ABB RAPID module: PointDesignationL.mod

MODULE PointDesignationL
     ! A point High enough so we prevent collision with right arm while counting the jars
    VAR robtarget HighPoint:=[[196.4363,403.2327,1110.746],[0.6038789,-0.03336211,0.3133152,0.7321549],[0,0,1,6],[-75.34075,9E+09,9E+09,9E+09,9E+09,9E+09]];

    ! Some points to move the jar from the corner of the orange station to it's place on the Black station
    CONST robtarget Mid_1:=[[554.8741,126.2235,262.6581],[0.1364978,0.4773159,0.8638731,-0.08521196],[0,0,1,4],[-114.2211,9E+09,9E+09,9E+09,9E+09,9E+09]];
    CONST robtarget Mid_2:=[[600.1525,126.022,252.2679],[0.2637084,-0.1631797,0.9305753,-0.194576],[0,-1,1,4],[-112.3011,9E+09,9E+09,9E+09,9E+09,9E+09]];
    CONST robtarget Mid_3:=[[477.903,13.94918,176.1371],[0.2316044,-0.2927044,0.7583622,-0.5343878],[0,-1,1,0],[-106.8015,9E+09,9E+09,9E+09,9E+09,9E+09]];
    CONST robtarget NearJar:=[[497.2253,-43.83931,99.90126],[0.3030509,-0.2875187,0.6406512,-0.6442509],[0,-1,1,0],[-97.47271,9E+09,9E+09,9E+09,9E+09,9E+09]];
    CONST robtarget AroundJar:=[[469.1461,57.8836,108.0806],[0.507771,-0.524942,0.4776943,-0.4882752],[0,2,1,0],[-104.2323,9E+09,9E+09,9E+09,9E+09,9E+09]];
    VAR   robtarget AroundJarTemp:=[[469.1461,57.8836,108.0806],[0.507771,-0.524942,0.4776943,-0.4882752],[0,2,1,0],[-104.2323,9E+09,9E+09,9E+09,9E+09,9E+09]];
    CONST robtarget AroundJar2:=[[542.9891,-82.73224,93.03219],[0.2985963,-0.3278764,0.6561838,-0.6105409],[0,-2,1,0],[-103.7693,9E+09,9E+09,9E+09,9E+09,9E+09]];
    CONST robtarget AroundJar2_whenreholdingB2ORNG:=[[469.1366,57.87084,77.23759],[0.507752,-0.5249463,0.4777046,-0.4882802],[0,2,1,0],[-108.5586,9E+09,9E+09,9E+09,9E+09,9E+09]];
    CONST robtarget AboveJar:=[[542.9725,-82.74228,181.6404],[0.2985748,-0.3278722,0.6561934,-0.6105433],[0,-2,1,0],[-103.7681,9E+09,9E+09,9E+09,9E+09,9E+09]];
    CONST robtarget AboveJarGripperClosed:=[[542.9536,-82.75277,130.0491],[0.2985461,-0.3278738,0.6561974,-0.6105522],[0,-2,1,0],[-103.7678,9E+09,9E+09,9E+09,9E+09,9E+09]];
    CONST robtarget AboveJarGripperClosedWithCover:=[[542.9536,-82.75277,133.5491],[0.2985461,-0.3278738,0.6561974,-0.6105522],[0,-2,1,0],[-103.7678,9E+09,9E+09,9E+09,9E+09,9E+09]];
    CONST robtarget Mid_4:=[[423.7296,10.00786,203.2406],[0.1999823,-0.2381262,0.7028769,-0.6397398],[0,-1,1,0],[-100.9323,9E+09,9E+09,9E+09,9E+09,9E+09]];
    CONST robtarget Mid_55:=[[399.0612,9.599308,227.3587],[0.09442355,0.1273759,0.7641647,-0.6252294],[0,-1,1,4],[-106.9641,9E+09,9E+09,9E+09,9E+09,9E+09]];
    CONST robtarget Mid_5:=[[294.4772,-31.24014,155.1631],[0.04340968,0.05411187,-0.7336182,0.6760117],[0,-1,1,0],[-88.41631,9E+09,9E+09,9E+09,9E+09,9E+09]];
    CONST robtarget Mid_6:=[[282.9144,9.219685,155.0747],[0.2976154,-0.2876453,-0.6585417,0.6284967],[0,0,1,0],[-89.4698,9E+09,9E+09,9E+09,9E+09,9E+09]];
    CONST robtarget AboveJarOnBlackStation:=[[300.4598,-108.7313,151.8091],[0.003938463,-0.003778499,-0.7494636,0.662023],[0,-1,1,0],[-106.3189,9E+09,9E+09,9E+09,9E+09,9E+09]];
    VAR  robtarget AboveJarOnBlackStationGripClosed:=[[297.6271,-108.8896,119.9425],[0.01007012,0.01952474,0.7378212,-0.6746386],[0,-1,1,0],[-86.27634,9E+09,9E+09,9E+09,9E+09,9E+09]];
    CONST robtarget AroundJarOnBlackStation:=[[300.4579,-108.7329,82.89008],[0.003940296,-0.003776616,-0.7494647,0.6620218],[0,-1,1,0],[-106.3195,9E+09,9E+09,9E+09,9E+09,9E+09]];
    VAR   robtarget AroundJarOnBlackStationTemp:=[[299.3644,-109.178,107.112],[0.02736216,0.0009125296,0.7063073,-0.7073758],[0,3,1,0],[-103.6667,9E+09,9E+09,9E+09,9E+09,9E+09]];
    CONST robtarget LiftComPos:=[[300.5263,-113.6614,67.16065],[0.002721211,-0.004066736,-0.7418641,0.6705323],[0,-1,1,0],[-105.7211,9E+09,9E+09,9E+09,9E+09,9E+09]];
    CONST robtarget JarLiftPositionSuc:=[[300.5102,-113.66146,171.1686],[0.0027393,-0.00406995,-0.7418638,0.6705326],[0,-1,1,0],[-105.7192,9E+09,9E+09,9E+09,9E+09,9E+09]];
    CONST robtarget JarLiftPositionFill:=[[300.4794,-113.6599,75.19614],[0.002774192,-0.004076869,-0.7418547,0.6705426],[0,-1,1,0],[-105.724,9E+09,9E+09,9E+09,9E+09,9E+09]];

    ! Points to take out nozzel if it get stucked (not emptied)
    CONST robtarget Mid_7:=[[370.2038,-32.87925,154.3524],[0.07468369,-0.01454502,-0.7141125,0.6958838],[0,-1,1,0],[-87.29718,9E+09,9E+09,9E+09,9E+09,9E+09]];
    CONST robtarget Mid_8:=[[298.1686,-36.30843,152.074],[0.4977928,-0.4529417,-0.5219991,0.5239877],[0,0,1,0],[-94.23718,9E+09,9E+09,9E+09,9E+09,9E+09]];
    CONST robtarget Mid_9:=[[186.6169,-50.05457,160.3339],[0.4734463,-0.4736413,-0.5224764,0.5277603],[0,0,1,0],[-91.6592,9E+09,9E+09,9E+09,9E+09,9E+09]];
    CONST robtarget Mid_10:=[[186.6181,-50.05502,140.333],[0.4734438,-0.4736429,-0.5224775,0.52776],[0,0,1,0],[-91.65925,9E+09,9E+09,9E+09,9E+09,9E+09]];
    CONST robtarget Mid_11:=[[186.5986,-50.04457,115.3932],[0.4734615,-0.4736465,-0.5224517,0.5277665],[0,0,1,0],[-102.8267,9E+09,9E+09,9E+09,9E+09,9E+09]];
    CONST robtarget Mid_12:=[[217.6369,12.78759,121.3941],[0.4734631,-0.4736456,-0.5224531,0.5277644],[0,0,1,0],[-102.8237,9E+09,9E+09,9E+09,9E+09,9E+09]];
    CONST robtarget Mid_13:=[[217.6287,67.39323,173.9318],[0.5328754,0.5396317,-0.4449165,-0.4763306],[0,0,-1,0],[-103.6128,9E+09,9E+09,9E+09,9E+09,9E+09]];
    CONST robtarget Mid_14:=[[74.23405,20.23655,236.8874],[0.5520811,0.5830978,-0.3836623,-0.4560775],[0,0,-1,0],[-103.5678,9E+09,9E+09,9E+09,9E+09,9E+09]];

    !points for opening jar lid by the right hand
    CONST robtarget OpenJarLidPoint:=[[438.2388,-72.98116,358.5548],[0.00297478,-0.001265666,0.7255163,-0.6881974],[1,3,1,4],[-105.4292,9E+09,9E+09,9E+09,9E+09,9E+09]];
    VAR   robtarget OpenJarLidPointTemp:=[[438.2388,-72.98116,358.5548],[0.00297478,-0.001265666,0.7255163,-0.6881974],[1,3,1,4],[-105.4292,9E+09,9E+09,9E+09,9E+09,9E+09]];
    VAR   robtarget Calibration_1:=[[299.3372,-109.1743,120.9315],[0.02733344,0.0009180704,0.7063079,-0.7073762],[0,3,1,0],[-103.664,9E+09,9E+09,9E+09,9E+09,9E+09]];

    !points For Held Jar in Hole Open And CLose
    CONST robtarget Held_AroundJarOnBlackStation:=[[299.3644,-109.178,82.112],[0.02736216,0.0009125296,0.7063073,-0.7073758],[0,3,1,0],[-103.6667,9E+09,9E+09,9E+09,9E+09,9E+09]];

    ! Point for the process: "PressToFill"
    VAR   robtarget PressToFill_1:=[[519.3063,24.34753,332.795],[0.02965483,-0.003819788,0.8239746,-0.5658373],[0,0,1,4],[-125.4765,9E+09,9E+09,9E+09,9E+09,9E+09]];
    VAR   robtarget PressToFill_2:=[[360.1791,-16.26686,468.5356],[0.02076531,0.07434192,-0.7122866,0.6976316],[0,1,-1,5],[-138.0943,9E+09,9E+09,9E+09,9E+09,9E+09]];
    VAR   robtarget PressToFill_3:=[[382.2147,-185.2293,384.7835],[0.04519064,0.01475611,-0.7181318,0.6942815],[0,1,-1,1],[-132.0769,9E+09,9E+09,9E+09,9E+09,9E+09]];
    VAR   robtarget PressToFill_4:=[[382.669,-190.6713,357.5512],[0.01741571,-0.005328834,-0.729151,0.6841105],[0,1,-1,1],[-128.3606,9E+09,9E+09,9E+09,9E+09,9E+09]];

!    VAR   robtarget PressToFill_33:=[[382.2147,-185.2293,384.7835],[0.04519064,0.01475611,-0.7181318,0.6942815],[0,1,-1,1],[-132.0769,9E+09,9E+09,9E+09,9E+09,9E+09]];
!    VAR   robtarget PressToFill_44:=[[382.2147,-185.2293,384.7835],[0.04519064,0.01475611,-0.7181318,0.6942815],[0,1,-1,1],[-132.0769,9E+09,9E+09,9E+09,9E+09,9E+09]];

    ! Point for the process: "PressToEmpty"
    VAR   robtarget PressToEmpty_1:=[[507.7589,-40.4017,439.5305],[0.05817171,-0.007579151,-0.7055872,0.7061907],[0,-1,1,4],[-114.2449,9E+09,9E+09,9E+09,9E+09,9E+09]];
    VAR   robtarget PressToEmpty_2:=[[409.6067,-92.53561,434.3977],[0.042205,0.04568755,-0.7053828,0.7060924],[0,-1,1,4],[-116.3767,9E+09,9E+09,9E+09,9E+09,9E+09]];
    VAR   robtarget PressToEmpty_3:=[[299.3842,-191.4462,440.1205],[0.05024188,-0.01052868,-0.7081174,0.7042263],[0,-1,1,4],[-127.8406,9E+09,9E+09,9E+09,9E+09,9E+09]];
    VAR   robtarget PressToEmpty_4:=[[293.096,-186.9429,416.2473],[0.07747618,-0.01482227,-0.7036266,0.706178],[0,-1,1,4],[-125.5751,9E+09,9E+09,9E+09,9E+09,9E+09]];

    ! Point for the process: "PressToDropNozzel"
    VAR   robtarget PressToDropNozzel_1:=[[461.1843,42.44297,476.7215],[0.06907275,-0.2256842,0.4523926,-0.8600212],[0,-1,1,4],[-111.1826,9E+09,9E+09,9E+09,9E+09,9E+09]];
    VAR   robtarget PressToDropNozzel_2:=[[372.7662,-47.38017,638.5932],[0.1921857,0.02402019,0.007670877,0.9810346],[0,-1,1,4],[-131.1653,9E+09,9E+09,9E+09,9E+09,9E+09]];
    VAR   robtarget PressToDropNozzel_3:=[[221.2352,-55.55732,540.6785],[0.4316385,-0.016244,0.01718291,0.9017367],[-2,-1,1,4],[-131.6921,9E+09,9E+09,9E+09,9E+09,9E+09]];
    VAR   robtarget PressToDropNozzel_4:=[[221.2341,-55.55516,525.4453],[0.4316393,-0.01624625,0.01718477,0.9017363],[-2,-1,1,4],[-131.6908,9E+09,9E+09,9E+09,9E+09,9E+09]];
! it was [233.9373,-54.62232,556.2691]

!    VAR   robtarget PressToDropNozzel_3:=[[256.4945,-57.30254,599.6307],[0.4860737,0.003330357,0.02276387,0.873615],[-1,-1,1,4],[-149.7138,9E+09,9E+09,9E+09,9E+09,9E+09]];
!    VAR   robtarget PressToDropNozzel_4:=[[233.9373,-54.62232,560.2691],[0.499564,-0.04660843,0.002983484,0.8650171],[-1,-1,1,4],[-152.252,9E+09,9E+09,9E+09,9E+09,9E+09]];

    VAR   robtarget TakeTheShit1:=[[634.1862,113.8697,192.1622],[0.3200693,-0.322839,0.6323941,-0.6272227],[-2,-1,1,4],[-99.01886,9E+09,9E+09,9E+09,9E+09,9E+09]];
    VAR   robtarget TakeTheShit2:=[[634.1827,-26.8355,192.1335],[0.3200635,-0.3228488,0.632426,-0.6271884],[-2,-2,1,4],[-104.1127,9E+09,9E+09,9E+09,9E+09,9E+09]];
    VAR   robtarget TakeTheShit3:=[[634.7637,-26.74809,100.5621],[0.3209175,-0.3231641,0.6328201,-0.6261914],[-2,-2,1,4],[-90.97301,9E+09,9E+09,9E+09,9E+09,9E+09]];
    VAR   robtarget TakeTheShit4:=[[233.9373,-54.62232,561.2691],[0.499564,-0.04660843,0.002983484,0.8650171],[-1,-1,1,4],[-152.252,9E+09,9E+09,9E+09,9E+09,9E+09]];
    VAR   robtarget TakeTheShit5:=[[233.9373,-54.62232,561.2691],[0.499564,-0.04660843,0.002983484,0.8650171],[-1,-1,1,4],[-152.252,9E+09,9E+09,9E+09,9E+09,9E+09]];
    VAR   robtarget TakeTheShit6:=[[233.9373,-54.62232,561.2691],[0.499564,-0.04660843,0.002983484,0.8650171],[-1,-1,1,4],[-152.252,9E+09,9E+09,9E+09,9E+09,9E+09]];
    VAR   robtarget TakeTheShit7:=[[233.9373,-54.62232,561.2691],[0.499564,-0.04660843,0.002983484,0.8650171],[-1,-1,1,4],[-152.252,9E+09,9E+09,9E+09,9E+09,9E+09]];
    VAR   robtarget TakeTheShit8:=[[233.9373,-54.62232,561.2691],[0.499564,-0.04660843,0.002983484,0.8650171],[-1,-1,1,4],[-152.252,9E+09,9E+09,9E+09,9E+09,9E+09]];

    !variables for pick_i_jar
    VAR robtarget temp11 := [[538.8864,-80.77894,221.9603],[0.006105556,-0.7083587,-0.7058232,-0.002063419],[0,1,0,0],[-143.5276,9E+09,9E+09,9E+09,9E+09,9E+09]];
    VAR robtarget temp22 := [[540.8173,-81.54366,142.0769],[0.01183519,-0.997568,-0.06846375,-0.005556368],[0,0,1,0],[-105.1789,9E+09,9E+09,9E+09,9E+09,9E+09]];
    VAR robtarget temp22_2 := [[538.8954,-80.79728,141.3239],[0.006108637,-0.708376,-0.7058056,-0.00213234],[0,1,0,0],[-143.5234,9E+09,9E+09,9E+09,9E+09,9E+09]];
    VAR robtarget temp33 := [[537.168,-23.01155,254.7484],[0.01269851,-0.9976652,-0.0668235,0.006131503],[0,1,1,0],[-137.7437,9E+09,9E+09,9E+09,9E+09,9E+09]];

    VAR robtarget temp111 := [[555.866,37.28145,260.7902],[0.003240219,0.515474,0.8375627,-0.1810106],[0,0,1,4],[-125.2034,9E+09,9E+09,9E+09,9E+09,9E+09]];

    ! points For EmptyJarInFunnel
    VAR robtarget EmptyJarInFunnel1 := [[542.9738,-82.7419,169.2278],[0.2985776,-0.3278701,0.6561945,-0.6105419],[0,-2,1,0],[-103.7685,9E+09,9E+09,9E+09,9E+09,9E+09]];
    VAR robtarget EmptyJarInFunnel2 := [[509.3815,-85.80142,333.4705],[0.2187517,-0.1670811,0.6963356,-0.6628335],[0,-1,1,4],[-120.4902,9E+09,9E+09,9E+09,9E+09,9E+09]];
    VAR robtarget EmptyJarInFunnel3 := [[522.1735,-69.93185,533.1119],[0.02160888,0.01557024,0.7216892,-0.6917046],[0,-1,0,4],[-131.8955,9E+09,9E+09,9E+09,9E+09,9E+09]];
    VAR robtarget EmptyJarInFunnel4 := [[579.168,-114.824,549.1523],[0.003460131,-0.01070567,0.7096465,-0.7044681],[0,-1,0,4],[-138.7548,9E+09,9E+09,9E+09,9E+09,9E+09]];
    VAR robtarget EmptyJarInFunnel5 := [[612.555,-124.0654,529.6832],[0.3797491,0.4447397,-0.5406042,0.604768],[0,-1,-1,4],[-138.8654,9E+09,9E+09,9E+09,9E+09,9E+09]];
    VAR jointtarget EmptyJarInFunnel6 := [[7.62782,-6.06867,-9.97302,-67.5133,48.472,-75.1432],[-11.3079,9E+09,9E+09,9E+09,9E+09,9E+09]];
    VAR robtarget EmptyJarInFunnel7 := [[639.8677,-123.5552,527.2377],[0.6505856,0.6549008,-0.1475849,0.3550521],[0,-1,-1,4],[-138.4516,9E+09,9E+09,9E+09,9E+09,9E+09]];
    VAR jointtarget EmptyJarInFunnel8 := [[7.62656,-4.88297,-12.1625,-71.4806,41.437,-137.477],[-12.4559,9E+09,9E+09,9E+09,9E+09,9E+09]];
!    VAR robtarget EmptyJarInFunnel1 := [[542.9738,-82.7419,169.2278],[0.2985776,-0.3278701,0.6561945,-0.6105419],[0,-2,1,0],[-103.7685,9E+09,9E+09,9E+09,9E+09,9E+09]];
!    VAR robtarget EmptyJarInFunnel2 := [[509.3815,-85.80142,333.4705],[0.2187517,-0.1670811,0.6963356,-0.6628335],[0,-1,1,4],[-120.4902,9E+09,9E+09,9E+09,9E+09,9E+09]];
!    VAR robtarget EmptyJarInFunnel3 := [[559.9003,-115.132,466.0972],[0.2435943,-0.18267,0.7031288,-0.6425756],[0,-1,1,4],[-135.0802,9E+09,9E+09,9E+09,9E+09,9E+09]];
!    VAR robtarget EmptyJarInFunnel4 := [[563.4829,-123.9325,453.4182],[0.1157927,-0.1737028,0.6953254,-0.6877077],[1,-1,1,4],[-101.6964,9E+09,9E+09,9E+09,9E+09,9E+09]];
!    VAR robtarget EmptyJarInFunnel5 := [[619.5551,-128.0116,495.3073],[0.09878946,0.2637755,-0.6589687,0.6974406],[1,-1,0,4],[-123.1754,9E+09,9E+09,9E+09,9E+09,9E+09]];
!    VAR jointtarget EmptyJarInFunnel6 := [[55.5188,-12.7313,-4.20476,-78.7748,51.5913,-66.4227],[-48.417,9E+09,9E+09,9E+09,9E+09,9E+09]];
!    VAR robtarget EmptyJarInFunnel7 := [[635.1245,-122.5695,495.139],[0.5098433,0.6154509,-0.3536144,0.4860419],[1,-1,-1,4],[-123.1736,9E+09,9E+09,9E+09,9E+09,9E+09]];
!    VAR jointtarget EmptyJarInFunnel8 := [[63.6341,-10.5993,-10.0918,-75.7709,53.0141,-103.894],[-55.7523,9E+09,9E+09,9E+09,9E+09,9E+09]];

    !points for TurnOnOffPump
    VAR robtarget TurnOnOffPump1 := [[526.153,38.09958,190.2548],[0.4197936,-0.5438984,0.5741237,-0.4453424],[0,-2,1,0],[-115.076,9E+09,9E+09,9E+09,9E+09,9E+09]];
    VAR robtarget TurnOnOffPump2 := [[606.993,68.08531,144.5578],[0.4903001,-0.5107632,0.4878295,-0.510636],[0,-2,1,0],[-115.457,9E+09,9E+09,9E+09,9E+09,9E+09]];
    VAR robtarget TurnOnOffPump3 := [[619.8333,69.28903,144.6728],[0.4774225,-0.5121061,0.5076672,-0.5020847],[0,-2,1,0],[-115.6113,9E+09,9E+09,9E+09,9E+09,9E+09]];
    VAR robtarget TurnOnOffPump4 := [[601.319,56.10294,144.9478],[0.4992474,-0.5128309,0.4744157,-0.5125294],[0,-2,1,0],[-117.0118,9E+09,9E+09,9E+09,9E+09,9E+09]];
    VAR robtarget TurnOnOffPump5 := [[620.4492,53.69436,144.059],[0.4864553,-0.5335312,0.4812441,-0.4971014],[0,-2,1,0],[-118.8294,9E+09,9E+09,9E+09,9E+09,9E+09]];

    !points to PutUsedFilterInPlate
    VAR robtarget PutUsedFilterInPlate1 := [[659.6804,294.5118,882.8145],[0.4583833,0.3134622,0.4479995,0.7006587],[1,1,1,4],[-84.16208,9E+09,9E+09,9E+09,9E+09,9E+09]];
    VAR robtarget PutUsedFilterInPlate2:= [[729.5361,316.8599,713.8459],[0.4743018,0.3458549,0.5544642,0.5899081],[-1,1,1,0],[-98.32429,9E+09,9E+09,9E+09,9E+09,9E+09]];
    VAR robtarget PutUsedFilterInPlate3 := [[627.6354,184.5434,403.376],[0.3160068,0.4302891,0.8267978,0.1771904],[-1,0,1,0],[-100.3993,9E+09,9E+09,9E+09,9E+09,9E+09]];
    VAR robtarget PutUsedFilterInPlate4 := [[693.8143,-76.36646,416.25],[0.4317127,0.4709601,0.739186,-0.2131308],[-1,0,1,4],[-144.9374,9E+09,9E+09,9E+09,9E+09,9E+09]];
    VAR robtarget PutUsedFilterInPlate5 := [[678.8909,-92.78428,400.3075],[0.4332832,0.4918353,0.7282541,-0.2000241],[-1,0,1,4],[-144.6771,9E+09,9E+09,9E+09,9E+09,9E+09]];
    VAR robtarget PutUsedFilterInPlate6 := [[675.0967,-96.8405,400.068],[0.4266095,0.459187,0.7422882,-0.2369805],[-1,0,1,4],[-144.0739,9E+09,9E+09,9E+09,9E+09,9E+09]];
    VAR robtarget PutUsedFilterInPlate7 := [[659.3943,-114.1817,416.0409],[0.433989,0.509519,0.6868571,-0.2833218],[-1,0,1,4],[-144.8195,9E+09,9E+09,9E+09,9E+09,9E+09]];
    VAR robtarget PutUsedFilterInPlate8 := [[660.7668,-108.0462,400.1559],[0.433766,0.5706262,0.6658683,-0.2070078],[-1,0,1,4],[-144.9431,9E+09,9E+09,9E+09,9E+09,9E+09]];
    VAR robtarget PutUsedFilterInPlate9_1 := [[653.9497,-117.6481,400.8684],[0.4377143,0.5433829,0.6762441,-0.2362946],[-1,0,1,4],[-144.7948,9E+09,9E+09,9E+09,9E+09,9E+09]];
    VAR robtarget PutUsedFilterInPlate9_2 := [[648.7224,-121.8801,400.2471],[0.4312582,0.5344699,0.6802632,-0.2561257],[-1,0,1,4],[-144.679,9E+09,9E+09,9E+09,9E+09,9E+09]];
    VAR robtarget PutUsedFilterInPlate9_3 := [[739.9978,-168.6412,416.739],[0.5754835,0.0372328,0.7205365,-0.3850449],[-2,0,1,5],[-176.9851,9E+09,9E+09,9E+09,9E+09,9E+09]];
    VAR robtarget PutUsedFilterInPlate9_4 := [[642.6837,-127.0515,399.5811],[0.4252243,0.525843,0.6833639,-0.2751133],[-1,0,1,4],[-144.6262,9E+09,9E+09,9E+09,9E+09,9E+09]];
    VAR robtarget PutUsedFilterInPlate10 := [[705.6974,15.20001,488.8885],[0.4072246,0.5465,0.6856457,-0.2557262],[-1,0,1,4],[-142.8558,9E+09,9E+09,9E+09,9E+09,9E+09]];
    VAR robtarget PutUsedFilterInPlate11 := [[540.3218,-77.23856,507.011],[0.6601061,0.1569522,0.7141562,-0.1720665],[-2,0,1,1],[-137.4751,9E+09,9E+09,9E+09,9E+09,9E+09]];
    VAR robtarget PutUsedFilterInPlate12 := [[520.2753,201.009,314.5901],[0.3981728,0.2501043,0.8246195,0.3144979],[-1,0,1,1],[-81.81605,9E+09,9E+09,9E+09,9E+09,9E+09]];
    VAR robtarget PutUsedFilterInPlate13 := [[685.7153,282.5469,791.6041],[0.3712364,0.4057675,0.3793415,0.7440674],[-1,0,1,1],[-85.34634,9E+09,9E+09,9E+09,9E+09,9E+09]];
    VAR robtarget PutUsedFilterInPlate14 := [[693.8467,-118.4703,438.5067],[0.5419858,0.1301268,0.7541113,-0.3473247],[-1,0,0,5],[-154.3998,9E+09,9E+09,9E+09,9E+09,9E+09]];

!    VAR robtarget PutUsedFilterInPlate1 := [[659.6804,294.5118,882.8145],[0.4583833,0.3134622,0.4479995,0.7006587],[1,1,1,4],[-84.16208,9E+09,9E+09,9E+09,9E+09,9E+09]];
!    VAR robtarget PutUsedFilterInPlate2:= [[729.5361,316.8599,713.8459],[0.4743018,0.3458549,0.5544642,0.5899081],[-1,1,1,0],[-98.32429,9E+09,9E+09,9E+09,9E+09,9E+09]];
!    VAR robtarget PutUsedFilterInPlate3 := [[627.6354,184.5434,403.376],[0.3160068,0.4302891,0.8267978,0.1771904],[-1,0,1,0],[-100.3993,9E+09,9E+09,9E+09,9E+09,9E+09]];
!    VAR robtarget PutUsedFilterInPlate4 := [[489.0176,30.28746,351.2016],[0.1877209,0.2861434,0.9252287,-0.1638134],[-1,0,1,0],[-103.505,9E+09,9E+09,9E+09,9E+09,9E+09]];
!    VAR robtarget PutUsedFilterInPlate5 := [[582.5636,-79.15766,464.9698],[0.4640646,0.1338722,0.8119465,-0.3278188],[-2,0,0,1],[-134.1977,9E+09,9E+09,9E+09,9E+09,9E+09]];
!    VAR robtarget PutUsedFilterInPlate6 := [[728.0447,-121.4309,437.2125],[0.5914922,0.08755949,0.7326388,-0.3251317],[-2,0,0,5],[-157.5888,9E+09,9E+09,9E+09,9E+09,9E+09]];
!    VAR robtarget PutUsedFilterInPlate7 := [[762.9458,-136.0914,431.3704],[0.5987817,0.06097189,0.7216019,-0.3421017],[-2,0,0,5],[-166.6636,9E+09,9E+09,9E+09,9E+09,9E+09]];
!    VAR robtarget PutUsedFilterInPlate8 := [[767.324,-138.3024,416.7769],[0.5755245,0.03726448,0.7204585,-0.3851265],[-2,1,0,5],[-176.9778,9E+09,9E+09,9E+09,9E+09,9E+09]];
!    VAR robtarget PutUsedFilterInPlate9_1 := [[753.6297,-152.0577,416.7436],[0.5754899,0.03723112,0.7205275,-0.3850524],[-2,0,0,5],[-176.9824,9E+09,9E+09,9E+09,9E+09,9E+09]];
!    VAR robtarget PutUsedFilterInPlate9_2 := [[749.1034,-159.2123,416.7399],[0.5754855,0.03723041,0.7205337,-0.3850474],[-2,0,0,5],[-176.9832,9E+09,9E+09,9E+09,9E+09,9E+09]];
!    VAR robtarget PutUsedFilterInPlate9_3 := [[739.9978,-168.6412,416.739],[0.5754835,0.0372328,0.7205365,-0.3850449],[-2,0,1,5],[-176.9851,9E+09,9E+09,9E+09,9E+09,9E+09]];
!    VAR robtarget PutUsedFilterInPlate9_4 := [[727.6697,-184.9677,416.7401],[0.575482,0.03723241,0.7205385,-0.3850435],[-2,0,1,5],[-176.9878,9E+09,9E+09,9E+09,9E+09,9E+09]];
!    VAR robtarget PutUsedFilterInPlate10 := [[716.1812,-180.2664,445.1152],[0.5987719,0.0609662,0.7216203,-0.3420811],[-2,0,1,5],[-166.6656,9E+09,9E+09,9E+09,9E+09,9E+09]];
!    VAR robtarget PutUsedFilterInPlate11 := [[540.3218,-77.23856,507.011],[0.6601061,0.1569522,0.7141562,-0.1720665],[-2,0,1,1],[-137.4751,9E+09,9E+09,9E+09,9E+09,9E+09]];
!    VAR robtarget PutUsedFilterInPlate12 := [[520.2753,201.009,314.5901],[0.3981728,0.2501043,0.8246195,0.3144979],[-1,0,1,1],[-81.81605,9E+09,9E+09,9E+09,9E+09,9E+09]];
!    VAR robtarget PutUsedFilterInPlate13 := [[685.7153,282.5469,791.6041],[0.3712364,0.4057675,0.3793415,0.7440674],[-1,0,1,1],[-85.34634,9E+09,9E+09,9E+09,9E+09,9E+09]];
!    VAR robtarget PutUsedFilterInPlate14 := [[693.8467,-118.4703,438.5067],[0.5419858,0.1301268,0.7541113,-0.3473247],[-1,0,0,5],[-154.3998,9E+09,9E+09,9E+09,9E+09,9E+09]];

    !Points for TwoPartsRemovingFilter
    VAR robtarget TwoPartsRemovingFilter1 := [[693.8467,-118.4703,438.5067],[0.5419858,0.1301268,0.7541113,-0.3473247],[-1,0,0,5],[-154.3998,9E+09,9E+09,9E+09,9E+09,9E+09]];
    VAR robtarget TwoPartsRemovingFilter2 := [[693.8467,-118.4703,438.5067],[0.5419858,0.1301268,0.7541113,-0.3473247],[-1,0,0,5],[-154.3998,9E+09,9E+09,9E+09,9E+09,9E+09]];
    VAR robtarget TwoPartsRemovingFilter3 := [[693.8467,-118.4703,438.5067],[0.5419858,0.1301268,0.7541113,-0.3473247],[-1,0,0,5],[-154.3998,9E+09,9E+09,9E+09,9E+09,9E+09]];
    VAR robtarget TwoPartsRemovingFilter4 := [[693.8467,-118.4703,438.5067],[0.5419858,0.1301268,0.7541113,-0.3473247],[-1,0,0,5],[-154.3998,9E+09,9E+09,9E+09,9E+09,9E+09]];
    VAR robtarget TwoPartsRemovingFilter5 := [[693.8467,-118.4703,438.5067],[0.5419858,0.1301268,0.7541113,-0.3473247],[-1,0,0,5],[-154.3998,9E+09,9E+09,9E+09,9E+09,9E+09]];
    VAR robtarget TwoPartsRemovingFilter6 := [[693.8467,-118.4703,438.5067],[0.5419858,0.1301268,0.7541113,-0.3473247],[-1,0,0,5],[-154.3998,9E+09,9E+09,9E+09,9E+09,9E+09]];
    VAR robtarget TwoPartsRemovingFilter7 := [[693.8467,-118.4703,438.5067],[0.5419858,0.1301268,0.7541113,-0.3473247],[-1,0,0,5],[-154.3998,9E+09,9E+09,9E+09,9E+09,9E+09]];
    VAR robtarget TwoPartsRemovingFilter8 := [[693.8467,-118.4703,438.5067],[0.5419858,0.1301268,0.7541113,-0.3473247],[-1,0,0,5],[-154.3998,9E+09,9E+09,9E+09,9E+09,9E+09]];

    ! Points for OpenLock
    VAR robtarget OpenLock1 := [[444.457,57.70416,428.058],[0.03391873,-0.7404301,-0.6687696,0.05796584],[0,0,1,4],[-130.1532,9E+09,9E+09,9E+09,9E+09,9E+09]];
    VAR robtarget OpenLock2 := [[395.5481,-18.01055,662.0746],[0.2859399,0.623473,0.6130692,-0.3920025],[0,0,0,4],[-175.4325,9E+09,9E+09,9E+09,9E+09,9E+09]];
    VAR robtarget OpenLock3 := [[140.0657,208.4361,815.2481],[0.7192939,0.5369508,0.3359022,-0.2854294],[-1,0,0,4],[-173.6447,9E+09,9E+09,9E+09,9E+09,9E+09]];
    VAR robtarget OpenLock4 := [[5.191932,227.3297,792.3666],[0.7067034,0.6950218,-0.1054061,-0.08002785],[-1,0,1,4],[-177.0995,9E+09,9E+09,9E+09,9E+09,9E+09]];
    VAR robtarget OpenLock5 := [[-0.2072967,211.4303,796.5233],[0.6647114,0.7327977,-0.1080445,-0.0974303],[0,0,1,4],[-174.9861,9E+09,9E+09,9E+09,9E+09,9E+09]];
    VAR robtarget OpenLock6 := [[18.56533,206.4703,803.4706],[0.5342917,0.7544999,-0.1925943,-0.3288917],[0,0,1,4],[174.4749,9E+09,9E+09,9E+09,9E+09,9E+09]];
    VAR robtarget OpenLock7 := [[26.01069,197.7451,805.874],[0.5572425,0.7538844,-0.1712465,-0.3030078],[0,0,1,4],[174.3886,9E+09,9E+09,9E+09,9E+09,9E+09]];
    VAR robtarget OpenLock8 := [[64.29567,196.4137,796.8171],[0.593984,0.7749357,-0.1077863,-0.1871893],[0,0,1,4],[174.6816,9E+09,9E+09,9E+09,9E+09,9E+09]];
    VAR robtarget OpenLock9 := [[141.9606,292.9066,771.1875],[0.6093736,0.7831045,0.0007116533,-0.1241395],[-1,0,1,4],[168.4337,9E+09,9E+09,9E+09,9E+09,9E+09]];
    VAR robtarget OpenDoor1 := [[9.252483,190.8387,946.1296],[0.5472443,0.4799712,-0.5484715,0.4114976],[0,0,2,4],[-170.3192,9E+09,9E+09,9E+09,9E+09,9E+09]];
    VAR robtarget OpenDoor2 := [[74.19608,109.5013,916.4993],[0.4329654,0.6321019,-0.5041171,0.398565],[0,0,2,4],[-170.9254,9E+09,9E+09,9E+09,9E+09,9E+09]];
    VAR robtarget OpenDoor3 := [[89.49784,107.546,916.007],[0.5552816,0.796127,-0.1462974,0.1908958],[0,0,1,4],[-171.0104,9E+09,9E+09,9E+09,9E+09,9E+09]];
    VAR robtarget OpenDoor4 := [[151.8988,-17.92328,903.7396],[0.6081921,0.7752277,-0.08229822,0.1495035],[0,0,1,4],[-165.7217,9E+09,9E+09,9E+09,9E+09,9E+09]];
    VAR robtarget OpenDoor5 := [[128.8867,-153.3557,902.482],[0.6733187,0.7204248,-0.1633569,0.03073454],[0,0,1,4],[172.9512,9E+09,9E+09,9E+09,9E+09,9E+09]];
    VAR robtarget OpenDoor6 := [[89.68587,-220.5704,903.4578],[0.6246813,0.7343436,0.08674885,-0.250973],[0,0,1,4],[-177.4566,9E+09,9E+09,9E+09,9E+09,9E+09]];
    VAR robtarget OpenDoor7 := [[75.34122,-242.0442,913.9324],[0.6577976,0.7158023,-0.01540221,-0.2338637],[0,0,1,4],[-178.3179,9E+09,9E+09,9E+09,9E+09,9E+09]];
    VAR robtarget OpenDoor8 := [[31.01233,-264.0635,919.3221],[0.6670828,0.6893996,-0.1408893,-0.2447015],[0,-1,1,4],[-174.4533,9E+09,9E+09,9E+09,9E+09,9E+09]];
    VAR robtarget OpenDoor9 := [[-22.00384,-264.0953,915.5707],[0.6219023,0.6198655,-0.2969985,-0.375228],[1,-1,2,4],[-179.6873,9E+09,9E+09,9E+09,9E+09,9E+09]];

    VAR num botNumber;

    VAR robtarget Error_TurnCtfg1 := [[170.2733,577.2457,243.9488],[0.00239963,0.3935039,-0.9193189,0.001257257],[1,-1,1,0],[-71.50956,9E+09,9E+09,9E+09,9E+09,9E+09]];
    VAR robtarget Error_TurnCtfg2 := [[-22.00384,-264.0953,915.5707],[0.6219023,0.6198655,-0.2969985,-0.375228],[1,-1,2,4],[-179.6873,9E+09,9E+09,9E+09,9E+09,9E+09]];
    VAR robtarget Error_TurnCtfg3 := [[-22.00384,-264.0953,915.5707],[0.6219023,0.6198655,-0.2969985,-0.375228],[1,-1,2,4],[-179.6873,9E+09,9E+09,9E+09,9E+09,9E+09]];

    VAR jointtarget shakeTubeClosed2 := [[3.84446,22.2276,18.0538,-143.954,79.6974,107.872],[24.8287,9E+09,9E+09,9E+09,9E+09,9E+09]];
    VAR jointtarget shakeTubeClosed3 := [[3.84446,22.2276,18.0538,-143.954,79.6974,107.872],[24.8287,9E+09,9E+09,9E+09,9E+09,9E+09]];

    VAR robtarget TightEquipping_1 := [[534.7612,-66.24588,448.1762],[0.0492238,0.994812,-0.08824188,0.01181438],[0,1,2,4],[-162.2959,9E+09,9E+09,9E+09,9E+09,9E+09]];
    VAR robtarget TightEquipping_2 := [[542.2573,-87.87419,378.4257],[0.01285309,-0.9964926,0.08052952,0.01876991],[0,1,1,0],[-166.3403,9E+09,9E+09,9E+09,9E+09,9E+09]];
    VAR robtarget TightEquipping_2_2 := [[541.673,-87.16678,340.6087],[0.004533053,0.9957977,-0.09128092,0.005848722],[0,1,1,0],[-156.5342,9E+09,9E+09,9E+09,9E+09,9E+09]];
    VAR robtarget TightEquipping_3 := [[541.676,-87.17374,325.7926],[0.004511012,0.9957966,-0.09129214,0.005883972],[0,1,1,0],[-156.5287,9E+09,9E+09,9E+09,9E+09,9E+09]];

    VAR robtarget PlaceFilterT1 := [[611.5538,188.9556,446.433],[0.4805578,-0.4926687,0.4904753,-0.53458],[0,-2,1,4],[-126.2647,9E+09,9E+09,9E+09,9E+09,9E+09]];
    VAR robtarget PlaceFilterT2 := [[630.3646,-3.842554,422.7774],[0.4727144,0.4460948,0.6930832,-0.3117309],[0,-1,1,4],[-127.4054,9E+09,9E+09,9E+09,9E+09,9E+09]];
    VAR robtarget PlaceFilterT3 := [[-53.30389,101.794,388.8003],[0.4561347,0.4681619,0.7094583,-0.2635043],[0,-1,1,4],[-128.3209,9E+09,9E+09,9E+09,9E+09,9E+09]];
    VAR robtarget PlaceFilterT4 := [[-47.41281,92.84719,385.8619],[0.4570908,0.4124958,0.7358824,-0.2817665],[0,-1,1,4],[-128.1705,9E+09,9E+09,9E+09,9E+09,9E+09]];
    VAR robtarget PlaceFilterT5 := [[-34.62054,96.09262,371.6744],[0.5329425,0.4002055,0.6885161,-0.2859257],[0,-1,2,4],[-123.7589,9E+09,9E+09,9E+09,9E+09,9E+09]];
    VAR robtarget PlaceFilterT6 := [[-51.12422,93.0301,363.8972],[0.5497394,0.4443694,0.6214367,-0.3378446],[0,-1,2,4],[-120.1642,9E+09,9E+09,9E+09,9E+09,9E+09]];
    VAR robtarget PlaceFilterT7 := [[-50.19769,79.45396,361.1102],[0.5492472,0.4124961,0.6310747,-0.3604431],[0,-1,2,4],[-120.3211,9E+09,9E+09,9E+09,9E+09,9E+09]];
    VAR robtarget PlaceFilterAbovePlate := [[-62.8074,56.11432,382.8491],[0.5123566,0.4925491,0.6392291,-0.2937214],[0,-1,2,4],[-127.7035,9E+09,9E+09,9E+09,9E+09,9E+09]];
    VAR robtarget PlaceFilterNearPlate := [[-45.5563,88.54259,396.3635],[0.5607795,0.3929399,0.6269881,-0.3714975],[0,-1,2,4],[-122.5446,9E+09,9E+09,9E+09,9E+09,9E+09]];
    VAR robtarget AwayFromPlate := [[-75.52215,109.7407,413.4696],[0.4992928,0.4945384,0.641796,-0.3069795],[0,-1,1,4],[-126.8027,9E+09,9E+09,9E+09,9E+09,9E+09]];
    VAR robtarget AboveTweezers := [[554.6125,187.2478,347.3214],[0.009141128,0.004833775,0.9999462,-0.0008103135],[1,0,0,4],[-91.82567,9E+09,9E+09,9E+09,9E+09,9E+09]];

    VAR robtarget TweezHelp1 := [[511.9012,185.3691,245.455],[0.2224359,-0.002102946,0.9749377,0.003773012],[2,-1,1,1],[-132.7921,9E+09,9E+09,9E+09,9E+09,9E+09]];

    VAR robtarget AboveTweezersReorient := [[558.8926,186.2785,147.8935],[0.221747,-0.007361691,0.975073,0.002584573],[1,0,1,1],[-112.0385,9E+09,9E+09,9E+09,9E+09,9E+09]];

    VAR robtarget AroundTweezersClose := [[567.4321,186.5397,219.4024],[0.4232465,0.006302222,0.9059864,0.003347539],[1,0,0,5],[-103.7297,9E+09,9E+09,9E+09,9E+09,9E+09]];
    VAR robtarget AroundTweezers := [[558.8488,186.2694,147.8692],[0.4070934,-0.004760375,0.9133582,0.005390874],[1,0,0,1],[-110.2104,9E+09,9E+09,9E+09,9E+09,9E+09]];
    VAR robtarget AroundTweezersGrip := [[558.4938,186.8937,134.9628],[0.009139122,0.00481677,0.9999463,-0.0008170585],[2,0,0,4],[-91.89567,9E+09,9E+09,9E+09,9E+09,9E+09]];


    VAR robtarget demonL1 := [[522.76,101.508,370.2567],[0.6395594,0.6600569,0.2778583,0.279434],[0,1,1,5],[-103.3218,9E+09,9E+09,9E+09,9E+09,9E+09]];
    VAR robtarget demonL2 := [[751.3519,323.1772,506.6777],[0.4281275,-0.6848934,0.4830146,-0.3381196],[0,0,-1,4],[-95.64716,9E+09,9E+09,9E+09,9E+09,9E+09]];


    VAR robtarget PickAndPlaceDoneAnalysisJars1 := [[537.182,-23.00752,254.7764],[0.01267209,-0.9976645,-0.06683949,0.006113062],[0,1,1,0],[-137.745,9E+09,9E+09,9E+09,9E+09,9E+09]];
    VAR robtarget PickAndPlaceDoneAnalysisJars2 := [[570.4759,125.5156,319.4925],[0.02538738,-0.9760913,-0.2154495,-0.0135202],[0,1,1,4],[-128.7419,9E+09,9E+09,9E+09,9E+09,9E+09]];
    VAR robtarget PickAndPlaceDoneAnalysisJars3 := [[540.7717,196.3669,306.0183],[0.2542661,-0.8990465,-0.2785631,-0.2224113],[0,1,1,4],[-127.332,9E+09,9E+09,9E+09,9E+09,9E+09]];
    VAR robtarget PickAndPlaceDoneAnalysisJars4 := [[525.423,188.4654,277.9547],[0.3815894,-0.5806725,0.5867504,-0.415852],[1,2,1,4],[-98.31242,9E+09,9E+09,9E+09,9E+09,9E+09]];
    VAR robtarget PickAndPlaceDoneAnalysisJars5 := [[561.7964,206.3241,252.4906],[0.3828885,-0.6013064,0.5689505,-0.4100272],[1,2,1,4],[-99.68642,9E+09,9E+09,9E+09,9E+09,9E+09]];
    VAR robtarget PickAndPlaceDoneAnalysisJars6 := [[655.5176,208.3491,209.3318],[0.3739311,-0.6130069,0.5491101,-0.4276402],[1,2,1,0],[-105.7962,9E+09,9E+09,9E+09,9E+09,9E+09]];
    VAR robtarget PickAndPlaceDoneAnalysisJars7 := [[525.423,188.4654,277.9547],[0.3815894,-0.5806725,0.5867504,-0.415852],[1,2,1,4],[-98.31242,9E+09,9E+09,9E+09,9E+09,9E+09]];
    VAR robtarget PickAndPlaceDoneAnalysisJars8 := [[587.5679,152.8891,234.2181],[0.4177889,-0.5915911,0.5426972,-0.4253847],[1,2,1,4],[-107.021,9E+09,9E+09,9E+09,9E+09,9E+09]];
    VAR robtarget PickAndPlaceDoneAnalysisJars9 := [[656.011,157.5958,208.3058],[0.4112938,-0.5956156,0.5396773,-0.4299162],[1,2,1,0],[-112.4389,9E+09,9E+09,9E+09,9E+09,9E+09]];
    VAR robtarget PickAndPlaceDoneAnalysisJars10 := [[525.423,188.4654,277.9547],[0.3815894,-0.5806725,0.5867504,-0.415852],[1,2,1,4],[-98.31242,9E+09,9E+09,9E+09,9E+09,9E+09]];

    !Points To Pick Jars From Their Station
    CONST robtarget Jar_i:=[[578.174,59.39053,136.758],[0.004271943,-0.9989691,-0.04503585,0.003779688],[-1,1,1,4],[-140.1295,9E+09,9E+09,9E+09,9E+09,9E+09]];
    VAR robtarget Jar_i_changing:=[[576.117,59.88061,138.5151],[0.001168195,-0.4148987,-0.9098623,0.002880127],[0,1,0,0],[-123.9672,9E+09,9E+09,9E+09,9E+09,9E+09]];
    CONST robtarget point_i:=[[576.1957,57.64332,274.0359],[0.0009735118,0.9987404,0.04927012,-0.009441065],[-1,1,1,4],[-140.0888,9E+09,9E+09,9E+09,9E+09,9E+09]];
    VAR robtarget point_i_changing:=[[575.8237,59.84186,160.0466],[0.001460813,-0.4148932,-0.9098634,0.003189074],[0,1,0,0],[-123.9444,9E+09,9E+09,9E+09,9E+09,9E+09]];
    ! Main MidPoint Of The System, abbreviated as "MMP"
    CONST robtarget MainMidPoint:=[[391.3701,138.0784,287.818],[0.01673144,-0.6788682,-0.7340627,-0.003146656],[0,0,1,4],[-105.6234,9E+09,9E+09,9E+09,9E+09,9E+09]];

    ! Centrifuge Center
    CONST robtarget CentrifugeCenter:=[[170.9407,572.1271,375.2909],[0.002034158,0.3950241,-0.9186674,0.001424496],[1,-1,1,0],[53.36959,9E+09,9E+09,9E+09,9E+09,9E+09]];

    ! Home of Left Arm
    CONST robtarget LeftArmHome:=[[-25.10183,35.87066,242.0362],[0.5241755,-0.456079,-0.4959679,0.5208146],[0,0,1,0],[-100.0034,9E+09,9E+09,9E+09,9E+09,9E+09]];
    CONST robtarget LeftArmHome2:=[[91.8348,42.58352,228.3557],[0.5194696,-0.447556,-0.5231068,0.5061662],[0,0,1,0],[-108.0553,9E+09,9E+09,9E+09,9E+09,9E+09]];

    ! Two points to rotate the Centrifuge rotor (axis)
    VAR jointtarget JointValuesAtRotationPoint := [[122.239,29.7559,-19.7606,-66.2785,71.2014,156.395],[3.56826,9E+09,9E+09,9E+09,9E+09,9E+09]];
    VAR jointtarget JointValuesAboveRotationPoint := [[119.561,28.2938,-22.0489,-67.2533,80.1595,74.3327],[13.3094,9E+09,9E+09,9E+09,9E+09,9E+09]];
    VAR jointtarget ApproachingPointAboveBlackSpot := [[106.568,30.0729,-17.8489,-77.2586,78.6877,35.8075],[28.6868,9E+09,9E+09,9E+09,9E+09,9E+09]];
    VAR jointtarget ApproachingPointAboveBlackSpot_2 := [[108.064,28.8972,-18.132,-76.5745,81.6513,35.4804],[29.6382,9E+09,9E+09,9E+09,9E+09,9E+09]];

    ! Points On The Path From MainMidPoint To Open Lid
    CONST robtarget FromMainMidPointToOpenLid1:=[[555.6271,255.7578,292.2513],[0.05483364,-0.590986,-0.8012478,-0.07570177],[0,0,1,4],[-108.0667,9E+09,9E+09,9E+09,9E+09,9E+09]];
    CONST robtarget FromMainMidPointToOpenLid2:=[[530.2897,361.5968,268.8058],[0.1494315,-0.5993652,-0.7668331,-0.174352],[0,1,1,4],[-100.0325,9E+09,9E+09,9E+09,9E+09,9E+09]];
    CONST robtarget FromMainMidPointToOpenLid3:=[[515.9312,467.775,263.5276],[0.03093584,0.1698122,0.935509,0.3082689],[0,0,0,4],[-80.93092,9E+09,9E+09,9E+09,9E+09,9E+09]];
    CONST robtarget FromMainMidPointToOpenLid4:=[[505.7648,470.2841,261.1846],[0.002194192,0.1675383,0.9377017,0.3043708],[0,0,0,4],[-81.04429,9E+09,9E+09,9E+09,9E+09,9E+09]];
    CONST robtarget StuckLidOpen1:=[[511.3714,387.8458,287.1512],[0.02826629,0.1820043,-0.9136657,-0.3623403],[1,0,0,4],[-71.72851,9E+09,9E+09,9E+09,9E+09,9E+09]];
    CONST robtarget StuckLidOpen2:=[[434.6936,360.7884,304.8413],[0.2318009,0.3091172,-0.7584912,-0.5247914],[2,0,0,4],[-53.44424,9E+09,9E+09,9E+09,9E+09,9E+09]];
    CONST robtarget StuckLidOpen3:=[[357.247,420.9841,302.484],[0.1812195,0.3416057,-0.7585484,-0.5244706],[2,0,0,4],[-46.24845,9E+09,9E+09,9E+09,9E+09,9E+09]];
    CONST robtarget StuckLidOpen4:=[[358.1856,425.442,389.0001],[0.04476143,0.5862212,-0.7014162,-0.4029348],[1,0,0,4],[-38.2786,9E+09,9E+09,9E+09,9E+09,9E+09]];
    CONST robtarget StuckLidOpen5:=[[332.1754,461.2852,492.5867],[0.08736742,-0.7816244,0.5270592,0.3219299],[1,0,0,4],[-8.962341,9E+09,9E+09,9E+09,9E+09,9E+09]];
    CONST robtarget StuckLidOpen6:=[[293.2359,466.8463,540.8222],[0.1258348,-0.8279678,0.4477544,0.3132907],[1,0,0,4],[5.271636,9E+09,9E+09,9E+09,9E+09,9E+09]];
    CONST robtarget StuckLidOpen7:=[[261.7409,484.2215,580.4375],[0.1996818,-0.8599576,0.3676526,0.2922871],[1,0,0,4],[19.18535,9E+09,9E+09,9E+09,9E+09,9E+09]];
    CONST robtarget StuckLidOpen8:=[[483.4654,510.2447,469.6231],[0.7102606,-0.5688905,0.09371739,-0.4038694],[0,2,1,4],[-106.5761,9E+09,9E+09,9E+09,9E+09,9E+09]];

    ! Points On The Path From MainMidPoint To the center of Centrifuge
    CONST robtarget FromMainMidPointToMidCtfg3:=[[450.2527,158.2175,451.6961],[0.01001458,0.6602603,0.7509692,-0.001124735],[1,0,1,4],[-82.61719,9E+09,9E+09,9E+09,9E+09,9E+09]];
    CONST robtarget FromMainMidPointToMidCtfg4:=[[323.9157,496.4598,484.945],[0.01640962,-0.2539656,0.9670679,-0.003446209],[1,-1,1,4],[20.83673,9E+09,9E+09,9E+09,9E+09,9E+09]];
    CONST robtarget FromMainMidPointToMidCtfg5:=[[210.4415,548.9407,460.6745],[0.001568333,0.3650672,-0.9308972,-0.01240387],[1,-1,1,0],[56.035,9E+09,9E+09,9E+09,9E+09,9E+09]];

    ! Points On The Path From MidCtfg To 0_angleHole
    CONST robtarget FromMidCtfg1To_0_angleHole1:=[[135.2472,548.4155,379.5739],[0.1102394,0.4009789,-0.9091622,0.02207327],[1,-1,1,0],[56.79922,9E+09,9E+09,9E+09,9E+09,9E+09]];
    CONST robtarget FromMidCtfg1To_0_angleHole2:=[[137.767,549.8556,345.9562],[0.1433132,0.3114628,-0.9385209,0.04038253],[1,-1,1,0],[30.70798,9E+09,9E+09,9E+09,9E+09,9E+09]];
    VAR   robtarget FromMidCtfg1To_0_angleHole3:=[[110.7217,535.2574,266.8914],[0.1269187,0.3825924,-0.9146844,0.02944688],[1,-1,1,0],[-98.19913,9E+09,9E+09,9E+09,9E+09,9E+09]];
    VAR   robtarget FromMidCtfg1To_0_angleHole3_New:=[[111.789,535.7997,267.7856],[0.1274696,0.3878011,-0.9109861,0.05887322],[1,-1,1,0],[-105.3579,9E+09,9E+09,9E+09,9E+09,9E+09]];

    ! Points On The Path From MidCtfg To 180_angleHole
    CONST robtarget FromMidCtfg1To_180_angleHole1:=[[204.7944,601.0034,381.2636],[0.1095933,-0.3805622,0.917484,0.03721399],[1,-1,1,0],[51.17107,9E+09,9E+09,9E+09,9E+09,9E+09]];
    CONST robtarget FromMidCtfg1To_180_angleHole2:=[[209.0023,611.7137,346.9704],[0.1469437,-0.2921586,0.9440864,0.04185314],[1,-1,1,0],[29.28295,9E+09,9E+09,9E+09,9E+09,9E+09]];
    VAR   robtarget FromMidCtfg1To_180_angleHole3:=[[223.1574,615.9135,260.1365],[0.1702223,-0.2959671,0.9375257,0.06688365],[1,-1,1,0],[-75.78754,9E+09,9E+09,9E+09,9E+09,9E+09]];
    VAR   robtarget FromMidCtfg1To_180_angleHole3_Ne:=[[227.1336,616.502,266.1725],[0.1514491,-0.3024495,0.9399686,0.04523797],[1,-1,1,0],[-65.41523,9E+09,9E+09,9E+09,9E+09,9E+09]];

    ! Points On The Path From Main mid-Point to rotate the Centrifuge
    CONST robtarget FromMainMidPointToRotCtfg1:=[[575.8081,255.8228,351.579],[0.01227518,-0.695172,-0.7186235,0.01286518],[1,0,1,4],[-89.50906,9E+09,9E+09,9E+09,9E+09,9E+09]];
    CONST robtarget FromMainMidPointToRotCtfg2:=[[567.9559,318.7068,381.2513],[0.02993935,-0.5620193,-0.8265089,-0.01100037],[1,0,1,4],[-75.64757,9E+09,9E+09,9E+09,9E+09,9E+09]];
    CONST robtarget FromMainMidPointToRotCtfg3:=[[525.4849,450.6662,230.9332],[0.08353104,0.1511458,0.9304417,0.3231961],[1,1,0,4],[-81.26004,9E+09,9E+09,9E+09,9E+09,9E+09]];
    CONST robtarget FromMainMidPointToRotCtfg4:=[[515.5418,457.6712,230.6592],[0.05555337,0.1403555,0.930378,0.3340823],[1,1,0,4],[-81.37067,9E+09,9E+09,9E+09,9E+09,9E+09]];

    ! Points On The Path From Main mid-Point to Closing point
    CONST jointtarget MidPointForClosing := [[28.2685,-33.041,-78.4157,41.7629,-6.42804,63.5832],[-9.81139,9E+09,9E+09,9E+09,9E+09,9E+09]];
    CONST robtarget ClosingPoint:=[[65.75471,516.1484,1045.955],[0.328339,-0.1202955,0.1630785,0.9225659],[0,2,-1,4],[-26.15103,9E+09,9E+09,9E+09,9E+09,9E+09]];

    ! Points On The Path From Last closing point to MMP
    CONST jointtarget FromLastClosingPointToMMP1 := [[90.4382,-25.79347,51.5233,75.0603,134.581,-97.955],[1.57864,9E+09,9E+09,9E+09,9E+09,9E+09]];

    ! Points On The Path From Main mid-Point to Picking first jar
    CONST robtarget PickFirstJar_1 := [[427.6173,92.83806,189.5824],[0.007409984,0.7110775,0.7029889,0.01097811],[0,1,0,4],[-113.2087,9E+09,9E+09,9E+09,9E+09,9E+09]];
    VAR   robtarget PickFirstJar_2 :=[[425.4446,92.12425,160.8428],[0.008086857,-0.7226321,-0.6911685,-0.004855193],[0,1,0,4],[-114.0697,9E+09,9E+09,9E+09,9E+09,9E+09]];
    VAR   robtarget PickFirstJar_2_New :=[[538.1926,95.65181,135.258],[0.001080828,0.7068843,0.7073284,-7.16987E-05],[0,1,1,0],[-116.1748,9E+09,9E+09,9E+09,9E+09,9E+09]];
    ! Points On The Path From Main mid-Point to Picking first jar
    CONST robtarget PickSecondJar_1 := [[423.384,165.8227,177.8916],[0.00139436,0.7509733,0.6602591,0.009747217],[0,1,1,4],[-107.2557,9E+09,9E+09,9E+09,9E+09,9E+09]];
    VAR   robtarget PickSecondJar_2 :=[[424.2891,164.7849,152.3529],[0.009089611,-0.7294349,-0.6839775,0.004105511],[0,1,1,4],[-107.7059,9E+09,9E+09,9E+09,9E+09,9E+09]];
    VAR   robtarget PickSecondJar_2_New :=[[572.6805,169.3293,135.3422],[0.003599708,0.7083769,0.7057958,0.006436796],[0,0,1,0],[-108.6508,9E+09,9E+09,9E+09,9E+09,9E+09]];
    !CLOSING LID POINTS
    CONST robtarget p21:=[[-54.21155,343.8949,967.5791],[0.006532962,0.005804455,0.3682394,-0.9296899],[0,2,-1,4],[24.1479,9E+09,9E+09,9E+09,9E+09,9E+09]];
    CONST robtarget p22:=[[-77.09963,449.7422,933.605],[0.06520384,-0.1339068,-0.206466,0.9670518],[0,2,-1,4],[17.39433,9E+09,9E+09,9E+09,9E+09,9E+09]];
    CONST robtarget p23:=[[-43.18761,468.7766,912.9921],[0.09353477,-0.1515866,-0.08896989,0.9799781],[0,2,-1,4],[18.28262,9E+09,9E+09,9E+09,9E+09,9E+09]];
    CONST robtarget p24:=[[41.73626,440.0399,839.5618],[0.148995,-0.1442001,-0.003190573,0.9782621],[1,2,-1,4],[6.475172,9E+09,9E+09,9E+09,9E+09,9E+09]];
    CONST robtarget p25:=[[86.86452,458.0172,764.6867],[0.1935159,-0.1626686,0.1153547,0.9606164],[1,2,-1,4],[-5.584281,9E+09,9E+09,9E+09,9E+09,9E+09]];
    CONST robtarget p26:=[[112.9737,409.2987,703.3761],[0.1068262,0.1209603,-0.1123169,-0.9804803],[1,1,-1,4],[20.20472,9E+09,9E+09,9E+09,9E+09,9E+09]];
    CONST robtarget p27:=[[173.5079,364.0509,627.8409],[0.1757005,0.05873886,-0.05200116,-0.9813129],[1,1,-1,4],[-41.145,9E+09,9E+09,9E+09,9E+09,9E+09]];
    CONST robtarget p28:=[[197.8417,349.8596,570.1074],[0.2092049,0.03806816,-0.03873761,-0.9763624],[1,1,-1,4],[-79.54709,9E+09,9E+09,9E+09,9E+09,9E+09]];
    CONST robtarget p29:=[[183.9448,358.7148,546.8412],[0.2329703,0.06726069,-0.07359605,-0.9673595],[1,1,-1,4],[-88.54404,9E+09,9E+09,9E+09,9E+09,9E+09]];
    CONST robtarget p210:=[[184.7424,360.5268,535.9896],[0.2401605,0.06532399,-0.07943761,-0.9652696],[1,1,-1,4],[-92.60441,9E+09,9E+09,9E+09,9E+09,9E+09]];
    CONST robtarget p211:=[[164.1227,305.8885,545.3433],[0.3675655,0.05272227,-0.0411719,-0.9275887],[1,1,-1,4],[-102.1549,9E+09,9E+09,9E+09,9E+09,9E+09]];
    CONST robtarget p212:=[[168.4138,314.394,537.3768],[0.35178,0.04191225,-0.05902426,-0.9332793],[1,1,-1,4],[-102.9348,9E+09,9E+09,9E+09,9E+09,9E+09]];

    ! Points For MoveFromCentrifugiToClosingPoint
    CONST robtarget p31:=[[165.8214,571.015,282.5802],[0.02916296,-0.954278,-0.2966616,-0.02224786],[-1,-1,-1,4],[-36.87019,9E+09,9E+09,9E+09,9E+09,9E+09]];
    CONST robtarget p32:=[[186.6241,584.8575,320.2978],[0.09885993,-0.9507332,-0.2937511,-0.006591114],[-1,-1,-1,4],[5.385326,9E+09,9E+09,9E+09,9E+09,9E+09]];
    CONST robtarget p33:=[[308.0265,567.2227,415.8525],[0.1808859,-0.9314811,-0.3084915,-0.06675492],[-1,-1,-1,0],[1.129918,9E+09,9E+09,9E+09,9E+09,9E+09]];
    CONST robtarget p34:=[[312.9203,463.9485,769.9877],[0.8306608,-0.5253688,0.005516294,0.1842822],[0,0,-1,0],[36.56224,9E+09,9E+09,9E+09,9E+09,9E+09]];
    CONST robtarget p35:=[[288.5476,366.4262,1040.767],[0.8106591,-0.070676,0.09136972,0.5740107],[0,0,-1,5],[116.7955,9E+09,9E+09,9E+09,9E+09,9E+09]];
    CONST robtarget p36:=[[-344.2679,148.036,986.1663],[0.2767537,-0.3358434,-0.08831543,0.8960006],[0,0,-1,5],[-161.1931,9E+09,9E+09,9E+09,9E+09,9E+09]];

    !REMOVE JARS FROM CENTRIFUGE POINTS
    CONST robtarget MidPoint1:=[[-15.36177,348.5852,335.8944],[0.01270505,-0.9236007,0.2928489,0.2470627],[-1,-1,0,4],[170.4837,9E+09,9E+09,9E+09,9E+09,9E+09]];
    CONST robtarget MidPoint2:=[[31.26853,436.978,413.9435],[0.04817061,-0.8782981,0.4121458,0.2375035],[-1,-1,0,4],[122.493,9E+09,9E+09,9E+09,9E+09,9E+09]];
    CONST robtarget MidPoint3:=[[111.0317,504.5747,448.034],[0.07192473,-0.7940943,0.5799018,0.1671973],[-1,-1,0,4],[90.6752,9E+09,9E+09,9E+09,9E+09,9E+09]];
    CONST robtarget MidPoint4:=[[165.9225,531.9565,411.8794],[0.0451835,-0.7357786,0.6625242,0.1328534],[-1,-1,0,4],[64.77802,9E+09,9E+09,9E+09,9E+09,9E+09]];
    CONST robtarget MidPoint5:=[[161.9857,546.8381,368.298],[0.01359276,-0.741698,0.6699201,0.03010476],[-1,-1,0,4],[60.27169,9E+09,9E+09,9E+09,9E+09,9E+09]];
    CONST robtarget MidPoint6:=[[151.0072,570.9579,331.5],[0.008055392,-0.7127928,0.7010313,0.02041362],[-1,-1,0,4],[57.89784,9E+09,9E+09,9E+09,9E+09,9E+09]];
    CONST robtarget MidPoint7:=[[174.8069,577.5685,314.3376],[0.004569697,-0.6978954,0.7161466,0.007425059],[-1,-1,0,4],[18.78571,9E+09,9E+09,9E+09,9E+09,9E+09]];
    CONST robtarget MidPoint8:=[[180.0738,545.2461,433.1544],[0.04159581,-0.7762719,0.6287719,0.01782117],[-1,-1,0,4],[70.30775,9E+09,9E+09,9E+09,9E+09,9E+09]];
    CONST robtarget MidPoint9:=[[164.01,552.978,413.8664],[0.03505084,-0.7764228,0.6292059,-0.006239605],[-1,-1,0,4],[67.89112,9E+09,9E+09,9E+09,9E+09,9E+09]];
    CONST robtarget MidPoint10:=[[191.7732,549.4138,428.0539],[0.01742604,0.6796587,-0.7243297,-0.1144856],[-1,-1,0,4],[36.42645,9E+09,9E+09,9E+09,9E+09,9E+09]];
    CONST robtarget MidPoint11:=[[197.9071,549.7495,404.888],[0.008835174,-0.8114156,0.5836176,0.03028545],[-1,-1,0,4],[39.40963,9E+09,9E+09,9E+09,9E+09,9E+09]];
    VAR robtarget PickingPoint:=[[169.4821,577.2805,403.2951],[0.001383028,-0.8565182,0.516115,0.0001807709],[0,2,0,5],[-29.27312,9E+09,9E+09,9E+09,9E+09,9E+09]];
    VAR robtarget PickingPoint2:=[[143.3968,519.1283,303.5095],[0.1127644,0.8357944,0.5214952,-0.1295168],[1,1,0,6],[-9.689839,9E+09,9E+09,9E+09,9E+09,9E+09]];
    CONST robtarget BlackSpotInsideCentrifuge:=[[169.4821,577.2805,382.2951],[0.001383028,-0.8565182,0.516115,0.0001807709],[0,2,0,5],[-29.27312,9E+09,9E+09,9E+09,9E+09,9E+09]];
    CONST robtarget temp:=[[239.1479,522.8867,309.5301],[0.09545279,0.9134718,-0.2259871,0.324635],[-1,-1,0,4],[-80.16695,9E+09,9E+09,9E+09,9E+09,9E+09]];

    ! Bottle handling points
    CONST robtarget bottleCommonHome:=[[467.4041,178.5938,237.3391],[0.0003125806,-0.9995312,0.02172055,0.02157629],[-1,0,2,0],[-88.23302,9E+09,9E+09,9E+09,9E+09,9E+09]];
    CONST robtarget bottleCommonTrans:=[[392.7921,23.88578,237.5083],[0.002209544,-0.9999967,-0.0003491008,-0.001229802],[-1,1,1,0],[-117.6451,9E+09,9E+09,9E+09,9E+09,9E+09]];
    CONST robtarget bottleCommonBase:=[[386.7303,-93.65413,117.2929],[0.002108854,-0.9999876,-0.004364781,-0.001148836],[0,1,1,0],[-117.5595,9E+09,9E+09,9E+09,9E+09,9E+09]];
    CONST robtarget bottleCommonAboveBase:=[[386.4107,-93.05679,185.3091],[0.002049777,-0.9999972,-0.0001199298,-0.001153563],[-1,1,1,0],[-117.4536,9E+09,9E+09,9E+09,9E+09,9E+09]];
    CONST robtarget bottle1Home:=[[480.8344,147.9202,113.9402],[0.007192627,0.9999054,-0.0116751,-0.001038288],[0,0,2,0],[-107.8764,9E+09,9E+09,9E+09,9E+09,9E+09]];
    CONST robtarget bottle1AboveHome:=[[478.707,147.0055,238.9896],[0.00712541,0.9999053,-0.01172807,-0.00101294],[-1,0,2,0],[-103.3061,9E+09,9E+09,9E+09,9E+09,9E+09]];
    CONST robtarget bottle2Home:=[[479.367,228.476,114.034],[0.0007215576,-0.9997553,0.02176413,0.00389439],[0,0,2,0],[-87.3568,9E+09,9E+09,9E+09,9E+09,9E+09]];
    CONST robtarget bottle2AboveHome:=[[479.3828,225.0841,225.2593],[0.0003531347,-0.9995302,0.02179706,0.02154359],[-1,0,2,0],[-85.76249,9E+09,9E+09,9E+09,9E+09,9E+09]];
   CONST robtarget bottle3Home:=[[398.3785,228.0408,114.4323],[0.0115562,-0.004664159,-0.9999208,-0.001770869],[0,-1,1,0],[-88.36855,9E+09,9E+09,9E+09,9E+09,9E+09]];
    CONST robtarget bottle3AboveHome:=[[402.2579,228.0397,205.5438],[0.01155248,-0.004658196,-0.9999209,-0.00175616],[-1,0,1,0],[-88.35867,9E+09,9E+09,9E+09,9E+09,9E+09]];
    CONST robtarget bottle1AnAboveHome:=[[563.0196,136.1761,332.199],[0.005840671,0.9999821,0.0009387526,0.0009419348],[-1,0,2,0],[-86.8104,9E+09,9E+09,9E+09,9E+09,9E+09]];
    CONST robtarget bottle1AnHome:=[[563.0155,136.1733,112.936],[0.005856541,0.9999819,0.0009519621,0.0009297157],[0,0,2,0],[-86.81136,9E+09,9E+09,9E+09,9E+09,9E+09]];
    CONST robtarget bottle2AnAboveHome:=[[563.0219,57.0204,363.5058],[0.005832558,0.9999821,0.0009283682,0.0009461052],[-1,0,2,0],[-86.81097,9E+09,9E+09,9E+09,9E+09,9E+09]];
    CONST robtarget bottle2AnHome:=[[564.9322,57.01807,115.4319],[0.001769608,0.9999943,-0.001265742,0.002560507],[0,0,2,0],[-86.81734,9E+09,9E+09,9E+09,9E+09,9E+09]];
    VAR robtarget bottleNumVar;
    VAR robtarget bottleNumVarAbove;
    CONST robtarget bottleCapAbove:=[[476.3817,38.13747,180.602],[0.007162502,0.999905,-0.0117312,-0.001027292],[-1,0,2,0],[-102.8574,9E+09,9E+09,9E+09,9E+09,9E+09]];
    CONST robtarget bottleCap:=[[476.3725,38.12706,47.16624],[0.007163816,0.9999049,-0.01173429,-0.001041268],[0,1,1,0],[-102.8565,9E+09,9E+09,9E+09,9E+09,9E+09]];

    VAR jointtarget JointValuesAboveRotationPoint1 := [[119.561,28.2938,-22.0489,-67.2533,80.1595,74.3327],[13.3094,9E+09,9E+09,9E+09,9E+09,9E+09]];
ENDMODULE
